{attribute 'linkalways'} 
{attribute 'no_explicit_call' := 'This FB is a CLASS and must be accessed using methods or properties'}
{attribute 'enable_dynamic_creation'}
FUNCTION_BLOCK _ETcVnContourRetrievalMode EXTENDS EnumDatatypeBase
VAR
	localData : ETcVnContourRetrievalMode;
	activeData : REFERENCE TO ETcVnContourRetrievalMode;
	enumBaseDatatype : _DINT(localData);
END_VAR

METHOD PRIVATE AddLocalEnumeration
VAR_INPUT
	Enumeration : T_MAXSTRING;
	Value : ETcVnContourRetrievalMode;
END_VAR
AddEnumeration(Enumeration, Value);
END_METHOD

PROPERTY PUBLIC Address : PVOID
GET
Address := ADR(activeData);
END_GET
END_PROPERTY

METHOD PUBLIC ClearReference
VAR_INPUT
END_VAR
activeData REF= localData;
SetBaseDatatypeReference();
END_METHOD

METHOD PUBLIC Clone : I_Datatype
VAR
    pClone : POINTER TO _ETcVnContourRetrievalMode;
END_VAR
pClone := __NEW(_ETcVnContourRetrievalMode(InitialValue := Value));
Clone := pClone^;
END_METHOD

METHOD FB_init : BOOL
VAR_INPUT
	bInitRetains : BOOL; // if TRUE, the retain variables are initialized (warm start / cold start)
	bInCopyCode : BOOL;  // if TRUE, the instance afterwards gets moved into the copy code (online change)
	InitialValue : ETcVnContourRetrievalMode;
END_VAR
localData := InitialValue;
AddBaseDatatype(enumBaseDatatype);
ClearReference();

AddLocalEnumeration('TCVN_CRM_EXTERNAL', ETcVnContourRetrievalMode.TCVN_CRM_EXTERNAL);
AddLocalEnumeration('TCVN_CRM_LIST', ETcVnContourRetrievalMode.TCVN_CRM_LIST);
AddLocalEnumeration('TCVN_CRM_CONNECTED_COMPONENTS', ETcVnContourRetrievalMode.TCVN_CRM_CONNECTED_COMPONENTS);
AddLocalEnumeration('TCVN_CRM_TREE', ETcVnContourRetrievalMode.TCVN_CRM_TREE);
AddLocalEnumeration('TCVN_CRM_FLOODFILL', ETcVnContourRetrievalMode.TCVN_CRM_FLOODFILL);
END_METHOD

PROPERTY PUBLIC Identifier : T_MAXSTRING
GET
Identifier := 'ETcVnContourRetrievalMode';
END_GET
END_PROPERTY

METHOD IsEnumeratorValueEqual : BOOL
VAR_INPUT
	Enumerator : I_KeyValueForwardEnumerator;
END_VAR
VAR
	storedValue : ETcVnContourRetrievalMode;
END_VAR
IF NOT Enumerator.TryGet(storedValue) THEN
	RETURN;
END_IF

IsEnumeratorValueEqual := storedValue = activeData;
END_METHOD

METHOD PUBLIC MakeReferenceTo
VAR_INPUT
	ReferenceTarget : REFERENCE TO ETcVnContourRetrievalMode;
END_VAR
activeData REF= ReferenceTarget;
SetBaseDatatypeReference();
END_METHOD

METHOD PROTECTED SetBaseDatatypeReference
VAR_INPUT
END_VAR
enumBaseDatatype.MakeReferenceTo(activeData);
END_METHOD

PROPERTY PUBLIC Size : UDINT
GET
Size := SIZEOF(activeData);
END_GET
END_PROPERTY

METHOD TryMakeReferenceTo : BOOL
VAR_INPUT
	Target : I_Datatype;
END_VAR
VAR
	pTargetData : POINTER TO ETcVnContourRetrievalMode;
END_VAR
IF NOT IsEquivalentTo(Target) THEN
	RETURN;
END_IF

pTargetData := Target.Address;
activeData REF= pTargetData^;
SetBaseDatatypeReference();
TryMakeReferenceTo := TRUE;
END_METHOD

PROPERTY PUBLIC Value : ETcVnContourRetrievalMode
GET
Value := activeData;
END_GET
SET
activeData := Value;
END_SET
END_PROPERTY

END_FUNCTION_BLOCK

(* stored: Version 1.1.0.1, ProductVersion 3.1.4024.13
   POU _ETcVnContourRetrievalMode: Id {a5ab3147-e9c7-098f-3ccb-c7a62b523d4e}, SpecialFunc None
   Folder Core: Id {22e770ae-f597-047d-2b07-5ae2eba7babd}
   Folder Protected: Id {4c6c47d5-a71a-0a73-1ecf-59912ce767ec}
   Folder Customize: Id {d80db340-a8cf-057f-11b1-2fc185bb9e7e}
   Folder Constructor: Id {e6e68511-a2f8-0498-0c96-f25258562f36}
   Folder Private: Id {d85bd196-9840-0a44-0684-9d291b906117}
   Folder Protected: Id {977c23bb-de1d-01a8-1d79-901a064127aa}
   Method AddLocalEnumeration: Id {237b5cb5-0092-041c-084d-25d346c4daff}
   Property Address: Id {dc7e3394-509c-060c-308e-522e52ed90f5}
   Get Get: Id {3df068e8-1bd6-09f0-2f9d-76758976c721}
   Method ClearReference: Id {bd79bb5a-88ce-0cdd-2c32-447c44bd9c44}
   Method Clone: Id {f2f8f34c-1372-0b93-35dc-dea8ce8b56e5}
   Method FB_init: Id {50a2e389-191f-0ba3-203b-a15b4e1f32a0}
   Property Identifier: Id {c6da98b2-9ff9-0438-3808-bb67fc9b3501}
   Get Get: Id {7ab0d653-cad4-0ab0-0c63-42eee9429e53}
   Method IsEnumeratorValueEqual: Id {eb28da45-58fe-0126-3221-be3cea6444c1}
   Method MakeReferenceTo: Id {e6c1a14e-cec2-052c-28c1-d56f5a4a2741}
   Method SetBaseDatatypeReference: Id {7488dc24-9995-0a25-23c0-c16f07de1d77}
   Property Size: Id {1028a8f1-475c-0473-13f5-41a82f8498a1}
   Get Get: Id {4d96c98d-0f9b-0aeb-04f5-862ce65eebc8}
   Method TryMakeReferenceTo: Id {96ceb65b-ed18-0ab5-2be8-94cd7cea5858}
   Property Value: Id {15a9a6f1-ae6c-0b44-126b-5d8ced8297bd}
   Get Get: Id {9f58c5df-94f1-00ad-3ca3-da3657aa3f18}
   Set Set: Id {02a825a0-ba1c-0aa6-1a04-512315cd30fe} *)
